// TIA Portal V19 export
TYPE "C406_VAR_IF_CAD_TYPIC"
   STRUCT
      BMO_HAND { ExternalAccessible := 'False'; ExternalVisible := 'False'; ExternalWritable := 'False'} : Bool;   // TRUE = CaDo in hand geschakeld FALSE = niet in hand
      STS_BEZ_TOE { ExternalAccessible := 'False'; ExternalVisible := 'False'; ExternalWritable := 'False'} : Bool;   // TRUE = Calamiteitendoorsteek bezig met beweging sluiten
      STS_BEZ_OPEN { ExternalAccessible := 'False'; ExternalVisible := 'False'; ExternalWritable := 'False'} : Bool;   // TRUE = Calamiteitendoorsteek bezig met beweging openen
      STS_POS_TOE { ExternalAccessible := 'False'; ExternalVisible := 'False'; ExternalWritable := 'False'} : Bool;   // TRUE = Calamiteitendoorsteek op stand Dicht
      STS_POS_OPEN { ExternalAccessible := 'False'; ExternalVisible := 'False'; ExternalWritable := 'False'} : Bool;   // TRUE = Calamiteitendoorsteek op stand Open
      STS_STOP { ExternalAccessible := 'False'; ExternalVisible := 'False'; ExternalWritable := 'False'} : Bool;   // TRUE = Calamiteitendoorsteek niet op een eindpositie en niet in beweging
      EXT_AUT { ExternalAccessible := 'False'; ExternalVisible := 'False'; ExternalWritable := 'False'} : Bool;   // Externe (hoofd) beveiliging aangesproken
      EXT_HW { ExternalAccessible := 'False'; ExternalVisible := 'False'; ExternalWritable := 'False'} : Bool;   // Sturings hardware (PLC) in storing
      STO { ExternalAccessible := 'False'; ExternalVisible := 'False'; ExternalWritable := 'False'} : Struct   // Opsomming van alle storingen en meldingen
         A001 : Bool;   // Beveiliging aangesproken
         A002 : Bool;   // Noodstop van de calamiteitendoorsteek is geactiveerd
         A003 : Bool;   // Storing calamiteitendoorsteek
         A004 : Bool;   // Algemene storing calamiteitendoorsteek
         A005 : Bool;   // Communicatie uitgevallen
         AT01 : Bool;   // Terugmelding Open niet tijdig bereikt
         AT02 : Bool;   // Terugmelding Dicht niet tijdig bereikt
         AT03 : Bool;   // Terugmeldingen Open en Dicht tegelijkertijd
         M001 : Bool;   // De calamiteitendoorsteek is afgekoppeld via de werkschakelaar
      END_STRUCT;
   END_STRUCT;
END_TYPE
